// TwinCAT 3 PLC project SPS
// ProgramVersion: 3.1.4026.10
// libraries:
//   Tc2_Standard, * (Beckhoff Automation GmbH)
//   Tc2_System, * (Beckhoff Automation GmbH)
//   Tc2_TcpIp, * (Beckhoff Automation GmbH)
// project tree:
//   DUTs/ REQUEST.TcDUT, REQUEST_.TcDUT, RESPONSE.TcDUT, RESPONSE_.TcDUT
//   GVLs/ GVL.TcGVL
//   / PlcTask.TcTTO
//   POUs/ Kommunikation_UDP.TcPOU, MAIN.TcPOU
// real-time tasks:
//   TASK PlcTask: cycle T#10ms, priority 20, ADS port 350
// I/O:
//   DEVICE Gerät 1 (RT-Ethernet Adapter)

CONFIGURATION SPS
    RESOURCE PLC ON TwinCAT3
        TASK PlcTask(INTERVAL := T#10ms, PRIORITY := 20);
        PROGRAM MAIN WITH PlcTask : MAIN;
    END_RESOURCE
END_CONFIGURATION

// ---- DUTs/REQUEST.TcDUT
TYPE REQUEST :
STRUCT
	Header			:UINT;		// Must be 0x1234
	Command			:UINT;		// Value according to the command table
	Data			:UDINT;		// data according to the actual command
END_STRUCT
END_TYPE

// ---- DUTs/REQUEST_.TcDUT
TYPE REQUEST_ :
STRUCT
	Command			:UINT;		// Value according to the command table
	Data			:ARRAY[0..18] OF UINT := [0];
END_STRUCT
END_TYPE

// ---- DUTs/RESPONSE.TcDUT
TYPE RESPONSE :
STRUCT
	HS_sequence			:UDINT;			// The sequence number of the current UDP record
	FT_sequence			:UDINT;			// The internal sample counter of the Compute Box
	Status				:UDINT;			// Status word of the sensor and Compute Box
	Fx					:UDINT;			// X-axis force in 32 bit Counts*
	Fy					:UDINT;			// Y-axis force in 32 bit Counts*
	Fz					:UDINT;			// Z-axis force in 32 bit Counts*
	Tx					:UDINT;			// X-axis torque in 32 bit Counts* (0 if not available)
	Ty					:UDINT;			// Y-axis torque in 32 bit Counts* (0 if not available)
	Tz					:UDINT;			// Z-axis torque in 32 bit Counts* (0 if not available)
END_STRUCT
END_TYPE

// ---- DUTs/RESPONSE_.TcDUT
TYPE RESPONSE_ :
STRUCT
	Header				:UINT;			// Fixed 0x1234
	Status				:UINT;			// Status word of the sensor and Compute Box
	Fx					:UINT;			// X-axis force in 32 bit Counts*
	Fy					:UINT;			// Y-axis force in 32 bit Counts*
	Fz					:UINT;			// Z-axis force in 32 bit Counts*
	Tx					:UINT;			// X-axis torque in 32 bit Counts* (0 if not available)
	Ty					:UINT;			// Y-axis torque in 32 bit Counts* (0 if not available)
	Tz					:UINT;			// Z-axis torque in 32 bit Counts* (0 if not available)
END_STRUCT
END_TYPE

// ---- GVLs/GVL.TcGVL
{attribute 'qualified_only'}
VAR_GLOBAL
	// Request
		Header			:UINT;			// Must be 0x1234
		Command			:UINT;			// Value according to the command table
		Data			:UINT;			// Value according to the command table
	
	// Response
		HS_sequence		:UINT;			// The sequence number of the current UDP record
		FT_sequence		:UINT;			// The internal sample counter of the Compute Box
		Status			:UINT;			// Status word of the sensor and Compute Box
		Fx				:UINT;			// X-axis force in 32 bit Counts*
		Fy				:UINT;			// Y-axis force in 32 bit Counts*
		Fz				:UINT;			// Z-axis force in 32 bit Counts*
		Tx				:UINT;			// X-axis torque in 32 bit Counts* (0 if not available)
		Ty				:UINT;			// Y-axis torque in 32 bit Counts* (0 if not available)
		Tz				:UINT;			// Z-axis torque in 32 bit Counts* (0 if not available)
		
END_VAR

// ---- POUs/MAIN.TcPOU
PROGRAM MAIN
VAR
	remotePort		:UDINT := 49151;
	remoteHost		:T_IPv4Addr := '192.168.1.1';
	
	stRemoteAddr 	: ST_SockAddr;
	
	Request			:REQUEST;
	Response		:RESPONSE;
	Request_		:REQUEST_;
	Response_		:RESPONSE_;
	
END_VAR
VAR_INPUT
	socket			:T_HSOCKET;
	
	Connect_busy	:BOOL;
	Connect_Done	:BOOL;
	
	Send_busy		:BOOL;
	Send_Done		:BOOL;
	
	Receive_busy	:BOOL;
	Receive_Done	:BOOL;
END_VAR

stRemoteAddr.sAddr := remoteHost;
stRemoteAddr.nPort := remotePort;

Request.Header 	:= 4660;
Request.Command	:= 2;
Request.Data := 1000;

Request_.Command := 0;



Kommunikation_UDP();

IF Connect_busy THEN
	Connect_Done := TRUE;
END_IF

IF Send_busy THEN
	Send_Done := TRUE;
END_IF

IF Receive_busy THEN
	Receive_Done := TRUE;
END_IF

END_PROGRAM

// ---- POUs/Kommunikation_UDP.TcPOU
PROGRAM Kommunikation_UDP
VAR
	Connect			:FB_SocketUdpCreate;
	Send			:FB_SocketUdpSendTo;
	Receive			:FB_SocketUdpReceiveFrom;
	
	Connect_		:FB_SocketConnect;
	Send_			:FB_SocketSend;
END_VAR

VAR_INPUT
	Receive_		:FB_SocketReceive;
END_VAR

Connect_(sRemoteHost := MAIN.stRemoteAddr.sAddr, nRemotePort := MAIN.stRemoteAddr.nPort); // FB_SocketConnect
Send_(hSocket := MAIN.socket, cbLen := SIZEOF(MAIN.Request_), pSrc := ADR(MAIN.Request_)); // FB_SocketSend
Connect(); // FB_SocketUdpCreate
MAIN.Connect_busy := Connect.bBusy;
Send(
    hSocket := MAIN.socket,
    sRemoteHost := MAIN.stRemoteAddr.sAddr,
    nRemotePort := MAIN.stRemoteAddr.nPort,
    cbLen := SIZEOF(MAIN.Request),
    pSrc := ADR(MAIN.Request)); // FB_SocketUdpSendTo
MAIN.Send_busy := Send.bBusy;
Receive_(hSocket := MAIN.socket, cbLen := SIZEOF(MAIN.Response_), pDest := ADR(MAIN.Response_)); // FB_SocketReceive
MAIN.Receive_busy := Receive_.bBusy;
MAIN.Connect_busy := Connect_.bBusy;
MAIN.Send_busy := Send_.bBusy;
Receive(hSocket := MAIN.socket, cbLen := SIZEOF(MAIN.Response), pDest := ADR(MAIN.Response)); // FB_SocketUdpReceiveFrom
MAIN.Receive_busy := Receive.bBusy;
MAIN.socket := Connect.hSocket;
MAIN.socket := Connect_.hSocket;

END_PROGRAM
